// TIA Portal V16 export
// export: Created 2021-11-12T13:31:52.6201346Z, ExportSetting WithDefaults, DisplayName Totally Integrated Automation Portal, DisplayVersion V16 Update 3, DisplayName TIA Portal Version Control Interface, DisplayVersion V16 Update 2, DisplayName TIA Portal Openness, DisplayVersion V16 Update 3, DisplayName SINAMICS Startdrive Advanced, DisplayVersion V16 Update 5, DisplayName SINAMICS Startdrive G130, G150, S120, S150, SINAMICS MV, S210, DisplayVersion V16 Update 5, DisplayName SINAMICS Startdrive G110M, G120, G120C, G120D, G120P, G115D, DisplayVersion V16 Update 5, DisplayName STEP 7 Professional, DisplayVersion V16 Update 3, DisplayName STEP 7 Safety, DisplayVersion V16, DisplayName WinCC UA Professional, DisplayVersion V16 Update 3
FUNCTION_BLOCK "Cab_000+UH10"   // FB29, LAD
TITLE = FB Cabinet V1.01
{ S7_Optimized_Access := 'TRUE' }
VERSION : 0.1
// MICE Wood block
// Cabinet V1.01
// functionality regarding cabinet, like errors from main switch, circuit breakers, temperature in cabinet,……
// stored: AutoNumber true, IsIECCheckEnabled false, IsRetainMemResEnabled false, MemoryReserve 100, SetENOAutomatically false, UDAEnableTagReadback false
   VAR
      SF_EC01_3_Alarm { S7_SetPoint := 'True'} : "STD_DI_Mon";
      SF_FC21_14_Alarm { S7_SetPoint := 'True'} : "STD_DI_Mon";
      SF_FC22_14_Alarm { S7_SetPoint := 'True'} : "STD_DI_Mon";
      SF_FB02_14_Alarm { S7_SetPoint := 'True'} : "STD_DI_Mon";
      SF_SF22_14_Alarm { S7_SetPoint := 'True'} : "STD_DI_Mon";
   END_VAR
   VAR_TEMP
      TB1Ack : Bool;
      TB1Aux : Bool;
   END_VAR
   VAR_TEMP   // added for the SCL form of the ladder/FBD networks
      _w1 : Bool;
      _w2 : Bool;
   END_VAR
BEGIN

REGION Network 1: Aknowledge logic - Any zone can acknowledge alarms
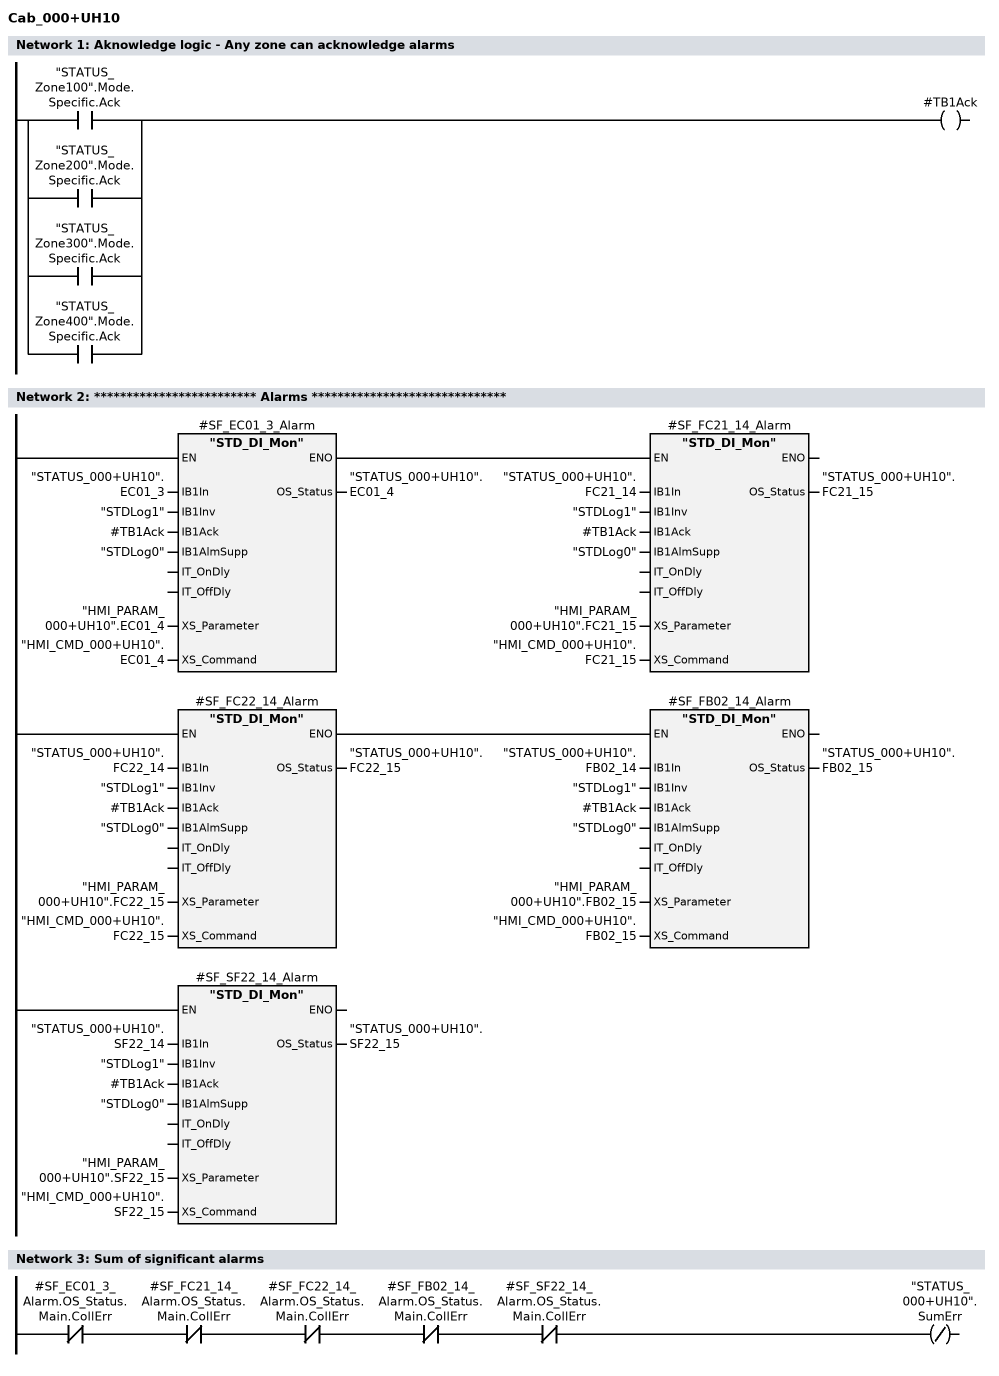
   RUNG wire#powerrail
      Contact( "STATUS_Zone100".Mode.Specific.Ack )
      wire#w1
      Coil( #TB1Ack )
   END_RUNG
   RUNG wire#powerrail
      Contact( "STATUS_Zone200".Mode.Specific.Ack )
   END_RUNG wire#w1
   RUNG wire#powerrail
      Contact( "STATUS_Zone300".Mode.Specific.Ack )
   END_RUNG wire#w1
   RUNG wire#powerrail
      Contact( "STATUS_Zone400".Mode.Specific.Ack )
   END_RUNG wire#w1
   // the same network as SCL:
   #TB1Ack := "STATUS_Zone100".Mode.Specific.Ack OR "STATUS_Zone200".Mode.Specific.Ack OR "STATUS_Zone300".Mode.Specific.Ack OR "STATUS_Zone400".Mode.Specific.Ack;
END_REGION

REGION Network 2: ************************* Alarms ******************************
   RUNG wire#powerrail
      #SF_EC01_3_Alarm(IB1In := "STATUS_000+UH10".EC01_3, IB1Inv := "STDLog1", IB1Ack := #TB1Ack, IB1AlmSupp := "STDLog0", IT_OnDly :=, IT_OffDly :=, XS_Parameter := "HMI_PARAM_000+UH10".EC01_4, XS_Command := "HMI_CMD_000+UH10".EC01_4, OS_Status => "STATUS_000+UH10".EC01_4)
      #SF_FC21_14_Alarm(IB1In := "STATUS_000+UH10".FC21_14, IB1Inv := "STDLog1", IB1Ack := #TB1Ack, IB1AlmSupp := "STDLog0", IT_OnDly :=, IT_OffDly :=, XS_Parameter := "HMI_PARAM_000+UH10".FC21_15, XS_Command := "HMI_CMD_000+UH10".FC21_15, OS_Status => "STATUS_000+UH10".FC21_15)
   END_RUNG
   RUNG wire#powerrail
      #SF_FC22_14_Alarm(IB1In := "STATUS_000+UH10".FC22_14, IB1Inv := "STDLog1", IB1Ack := #TB1Ack, IB1AlmSupp := "STDLog0", IT_OnDly :=, IT_OffDly :=, XS_Parameter := "HMI_PARAM_000+UH10".FC22_15, XS_Command := "HMI_CMD_000+UH10".FC22_15, OS_Status => "STATUS_000+UH10".FC22_15)
      #SF_FB02_14_Alarm(IB1In := "STATUS_000+UH10".FB02_14, IB1Inv := "STDLog1", IB1Ack := #TB1Ack, IB1AlmSupp := "STDLog0", IT_OnDly :=, IT_OffDly :=, XS_Parameter := "HMI_PARAM_000+UH10".FB02_15, XS_Command := "HMI_CMD_000+UH10".FB02_15, OS_Status => "STATUS_000+UH10".FB02_15)
   END_RUNG
   RUNG wire#powerrail
      #SF_SF22_14_Alarm(IB1In := "STATUS_000+UH10".SF22_14, IB1Inv := "STDLog1", IB1Ack := #TB1Ack, IB1AlmSupp := "STDLog0", IT_OnDly :=, IT_OffDly :=, XS_Parameter := "HMI_PARAM_000+UH10".SF22_15, XS_Command := "HMI_CMD_000+UH10".SF22_15, OS_Status => "STATUS_000+UH10".SF22_15)
   END_RUNG
   // the same network as SCL:
   #SF_EC01_3_Alarm(IB1In := "STATUS_000+UH10".EC01_3,   // "STD_DI_Mon"
                    IB1Inv := "STDLog1",
                    IB1Ack := #TB1Ack,
                    IB1AlmSupp := "STDLog0",
                    XS_Parameter := "HMI_PARAM_000+UH10".EC01_4,
                    XS_Command := "HMI_CMD_000+UH10".EC01_4,
                    OS_Status => "STATUS_000+UH10".EC01_4,
                    ENO => #_w1);
   IF #_w1 THEN
       #SF_FC21_14_Alarm(IB1In := "STATUS_000+UH10".FC21_14,   // "STD_DI_Mon"
                         IB1Inv := "STDLog1",
                         IB1Ack := #TB1Ack,
                         IB1AlmSupp := "STDLog0",
                         XS_Parameter := "HMI_PARAM_000+UH10".FC21_15,
                         XS_Command := "HMI_CMD_000+UH10".FC21_15,
                         OS_Status => "STATUS_000+UH10".FC21_15);
   END_IF;
   #SF_FC22_14_Alarm(IB1In := "STATUS_000+UH10".FC22_14,   // "STD_DI_Mon"
                     IB1Inv := "STDLog1",
                     IB1Ack := #TB1Ack,
                     IB1AlmSupp := "STDLog0",
                     XS_Parameter := "HMI_PARAM_000+UH10".FC22_15,
                     XS_Command := "HMI_CMD_000+UH10".FC22_15,
                     OS_Status => "STATUS_000+UH10".FC22_15,
                     ENO => #_w2);
   IF #_w2 THEN
       #SF_FB02_14_Alarm(IB1In := "STATUS_000+UH10".FB02_14,   // "STD_DI_Mon"
                         IB1Inv := "STDLog1",
                         IB1Ack := #TB1Ack,
                         IB1AlmSupp := "STDLog0",
                         XS_Parameter := "HMI_PARAM_000+UH10".FB02_15,
                         XS_Command := "HMI_CMD_000+UH10".FB02_15,
                         OS_Status => "STATUS_000+UH10".FB02_15);
   END_IF;
   #SF_SF22_14_Alarm(IB1In := "STATUS_000+UH10".SF22_14,   // "STD_DI_Mon"
                     IB1Inv := "STDLog1",
                     IB1Ack := #TB1Ack,
                     IB1AlmSupp := "STDLog0",
                     XS_Parameter := "HMI_PARAM_000+UH10".SF22_15,
                     XS_Command := "HMI_CMD_000+UH10".SF22_15,
                     OS_Status => "STATUS_000+UH10".SF22_15);
END_REGION

REGION Network 3: Sum of significant alarms
   RUNG wire#powerrail
      I_Contact( #SF_EC01_3_Alarm.OS_Status.Main.CollErr )
      I_Contact( #SF_FC21_14_Alarm.OS_Status.Main.CollErr )
      I_Contact( #SF_FC22_14_Alarm.OS_Status.Main.CollErr )
      I_Contact( #SF_FB02_14_Alarm.OS_Status.Main.CollErr )
      I_Contact( #SF_SF22_14_Alarm.OS_Status.Main.CollErr )
      I_Coil( "STATUS_000+UH10".SumErr )
   END_RUNG
   // the same network as SCL:
   "STATUS_000+UH10".SumErr := NOT (NOT #SF_EC01_3_Alarm.OS_Status.Main.CollErr AND NOT #SF_FC21_14_Alarm.OS_Status.Main.CollErr AND NOT #SF_FC22_14_Alarm.OS_Status.Main.CollErr AND NOT #SF_FB02_14_Alarm.OS_Status.Main.CollErr AND NOT #SF_SF22_14_Alarm.OS_Status.Main.CollErr);
END_REGION

REGION Network 4: Significant voltage OK
END_REGION
END_FUNCTION_BLOCK
